// TwinCAT 3 PLC project tmo_spectrometer_motion
// ProgramVersion: 3.1.4022.7
// libraries:
//   lcls-twincat-motion, * (SLAC)
//   Tc2_MC2, * (Beckhoff Automation GmbH)
//   Tc2_Standard, * (Beckhoff Automation GmbH)
//   Tc2_System, * (Beckhoff Automation GmbH)
//   Tc2_Utilities, * (Beckhoff Automation GmbH)
//   Tc3_Module, * (Beckhoff Automation GmbH)
// project tree:
//   GVLs/ IO.TcGVL
//   / PlcTask.TcTTO
//   POUs/ Main.TcPOU
// real-time tasks:
//   TASK PlcTask: cycle T#10ms, priority 20, ADS port 350
// motion (NC):
//   TASK NC-Task 1 SAF: cycle T#2ms, priority 4, ADS port 501
//   TASK NC-Task 1 SVB: cycle T#10ms, priority 8, ADS port 511
//   AXIS LensX (id 1)
//     Dynamic: Acceleration=2, Deceleration=2
//     Velo: SlowManual=0.1, FastManual=1, Maximum=1
//     OtherSettings: AllowMotionCmdToSlave=true, PulseDistancePos=0.5, PulseDistanceNeg=0.5
//     encoder EncType=4
//       EncPara: ScaleFactorNumerator=3.90625e-05, MaxCount=#x0000ffff
//         Inc: RefSoftSyncMask=#x0000ffff
//     drive DrvType=24
//       Analog: VeloReferenz=4.5, ScaleFactorActTorque=0.1
//       TimeComp: TaskDelayCycles=1
//     controller CtrType=2
//       CtrPara: PriorControlFactor=1
//         PosDiffControl: Range=1
//         Observer: BandWidth=20
//   AXIS FoilX (id 2)
//     Dynamic: Acceleration=2, Deceleration=2
//     Velo: SlowManual=0.1, FastManual=1, Maximum=1
//     OtherSettings: AllowMotionCmdToSlave=true, PulseDistancePos=0.5, PulseDistanceNeg=0.5
//     encoder EncType=4
//       EncPara: ScaleFactorNumerator=0.000244140625, MaxCount=#x0000ffff
//         SoftEndMaxControl: Enable=true, Range=-1
//         Inc: RefSoftSyncMask=#x0000ffff
//     drive DrvType=24
//       Analog: VeloReferenz=31.25, ScaleFactorActTorque=0.1
//       TimeComp: TaskDelayCycles=1
//     controller CtrType=2
//       CtrPara: PriorControlFactor=1
//         PosDiffControl: Range=1
//         Observer: BandWidth=20
//   AXIS ZonePlateX (id 3)
//     Dynamic: Acceleration=2, Deceleration=2
//     Velo: SlowManual=0.1, FastManual=1, Maximum=1
//     OtherSettings: AllowMotionCmdToSlave=true, PulseDistancePos=0.5, PulseDistanceNeg=0.5
//     encoder EncType=4
//       EncPara: ScaleFactorNumerator=0.000103125, Inverse=true, MaxCount=#x0000ffff
//         Inc: RefSoftSyncMask=#x0000ffff
//     drive DrvType=24
//       DrvPara: Inverse=true
//         Analog: VeloReferenz=13.2, ScaleFactorActTorque=0.1
//         TimeComp: TaskDelayCycles=1
//     controller CtrType=2
//       CtrPara: PriorControlFactor=1
//         PosDiffControl: Range=1
//         Observer: BandWidth=20
//   AXIS ZonePlateY (id 4)
//     Dynamic: Acceleration=2, Deceleration=2
//     Velo: SlowManual=0.1, FastManual=1, Maximum=1
//     OtherSettings: AllowMotionCmdToSlave=true, PulseDistancePos=0.5, PulseDistanceNeg=0.5
//     encoder EncType=4
//       EncPara: ScaleFactorNumerator=4.6875e-05, MaxCount=#x0000ffff
//         Inc: RefSoftSyncMask=#x0000ffff
//     drive DrvType=24
//       Analog: VeloReferenz=6, ScaleFactorActTorque=0.1
//       TimeComp: TaskDelayCycles=1
//     controller CtrType=2
//       CtrPara: PriorControlFactor=1
//         PosDiffControl: Range=1
//         Observer: BandWidth=20
//   AXIS ZonePlateZ (id 5)
//     Dynamic: Acceleration=2, Deceleration=2
//     Velo: SlowManual=0.1, FastManual=1, Maximum=1
//     OtherSettings: AllowMotionCmdToSlave=true, PulseDistancePos=0.5, PulseDistanceNeg=0.5
//     encoder EncType=4
//       EncPara: ScaleFactorNumerator=7.8125e-05, ScaleFactorDenominator=1.6, MaxCount=#x0000ffff
//         Inc: RefSoftSyncMask=#x0000ffff
//     drive DrvType=24
//       Analog: VeloReferenz=6.25, ScaleFactorActTorque=0.1
//       TimeComp: TaskDelayCycles=1
//     controller CtrType=2
//       CtrPara: PriorControlFactor=1
//         PosDiffControl: Range=1
//         Observer: BandWidth=20
//   AXIS YagX (id 6)
//     Dynamic: Acceleration=2, Deceleration=2
//     Velo: SlowManual=0.1, FastManual=1, Maximum=1
//     OtherSettings: AllowMotionCmdToSlave=true, PulseDistancePos=0.5, PulseDistanceNeg=0.5
//     encoder EncType=4
//       EncPara: ScaleFactorNumerator=7.8125e-05, Inverse=true, MaxCount=#x0000ffff
//         Inc: RefSoftSyncMask=#x0000ffff
//     drive DrvType=24
//       DrvPara: Inverse=true
//         Analog: VeloReferenz=10, ScaleFactorActTorque=0.1
//         TimeComp: TaskDelayCycles=1
//     controller CtrType=2
//       CtrPara: PriorControlFactor=1
//         PosDiffControl: Range=1
//         Observer: BandWidth=20
//   AXIS YagY (id 7)
//     Dynamic: Acceleration=2, Deceleration=2
//     Velo: SlowManual=0.1, FastManual=1, Maximum=1
//     OtherSettings: AllowMotionCmdToSlave=true, PulseDistancePos=0.5, PulseDistanceNeg=0.5
//     encoder EncType=4
//       EncPara: ScaleFactorNumerator=7.8125e-05, MaxCount=#x0000ffff
//         Inc: RefSoftSyncMask=#x0000ffff
//     drive DrvType=24
//       Analog: VeloReferenz=10, ScaleFactorActTorque=0.1
//       TimeComp: TaskDelayCycles=1
//     controller CtrType=2
//       CtrPara: PriorControlFactor=1
//         PosDiffControl: Range=1
//         Observer: BandWidth=20
//   AXIS YagZ (id 8)
//     Dynamic: Acceleration=2, Deceleration=2
//     Velo: SlowManual=0.1, FastManual=1, Maximum=1
//     OtherSettings: AllowMotionCmdToSlave=true, PulseDistancePos=0.5, PulseDistanceNeg=0.5
//     encoder EncType=4
//       EncPara: ScaleFactorNumerator=9.6875e-05, Inverse=true, MaxCount=#x0000ffff
//         Inc: RefSoftSyncMask=#x0000ffff
//     drive DrvType=24
//       DrvPara: Inverse=true
//         Analog: VeloReferenz=12.7, ScaleFactorActTorque=0.1
//         TimeComp: TaskDelayCycles=1
//     controller CtrType=2
//       CtrPara: PriorControlFactor=1
//         PosDiffControl: Range=1
//         Observer: BandWidth=20
//   AXIS YagTheta (id 9)
//     Dynamic: Acceleration=2, Deceleration=2
//     Velo: SlowManual=0.1, FastManual=1, Maximum=1
//     OtherSettings: AllowMotionCmdToSlave=true, PulseDistancePos=0.5, PulseDistanceNeg=0.5
//     encoder EncType=4
//       EncPara: ScaleFactorNumerator=1.171875e-05, ScaleFactorDenominator=0.036667, MaxCount=#x0000ffff
//         Inc: RefSoftSyncMask=#x0000ffff
//     drive DrvType=24
//       Analog: VeloReferenz=409.0905372, ScaleFactorActTorque=0.1
//       TimeComp: TaskDelayCycles=1
//     controller CtrType=2
//       CtrPara: PriorControlFactor=1
//         PosDiffControl: Range=1
//         Observer: BandWidth=20
// I/O:
//   DEVICE Device 1 (EtherCAT), AmsNetId 172.21.132.142.2.1
//     Term 19 (EK1200) [EK1200-5000 EtherCAT Power supply (2A E-Bus)]
//       Term 20 (EL2202) [EL2202 2Ch. Dig. Output 24V, 0.5A]
//       Term 21 (EL6070) [EL6070 1Ch. Licensing-Terminal]
//       Term 22 (EL6695) [EL6695 EtherCAT Bridge terminal (Primary)]
//       Term 23 (EK1122) [EK1122 2 port EtherCAT junction]
//         Term 24 (EK1100) [EK1100 EtherCAT Coupler (2A E-Bus)]
//           EL7031-LensX [EL7031 1Ch. Stepper motor output stage (24V, 1.5A)]
//           LensX_EL1004
//           FoilX-EL7041 [EL7041 1Ch. Stepper motor output stage (50V, 5A)]
//           ZonePlateX-EL7041 [EL7041 1Ch. Stepper motor output stage (50V, 5A)]
//           ZonePlateY-EL7041 [EL7041 1Ch. Stepper motor output stage (50V, 5A)]
//           ZonePlateZ-EL7041 [EL7041 1Ch. Stepper motor output stage (50V, 5A)]
//           YagX-EL7041 [EL7041 1Ch. Stepper motor output stage (50V, 5A)]
//           YagY-EL7041 [EL7041 1Ch. Stepper motor output stage (50V, 5A)]
//           YagZ-EL7041 [EL7041 1Ch. Stepper motor output stage (50V, 5A)]
//           YagTheta-EL7041 [EL7041 1Ch. Stepper motor output stage (50V, 5A)]
//           Term 35 (EL9011) [EL9011 End Terminal]
// variable links:
//   (this object) <-> Device 1 (EtherCAT)/Term 19 (EK1200)/Term 23 (EK1122)/Term 24 (EK1100)/EL7031-LensX
//     Drive/Inputs/In/nState1 @bit 3 <-> STM Status/Status/Error
//     Drive/Inputs/In/nState1 @bit 5 <-> STM Status/Status/Moving negative
//     Drive/Inputs/In/nState1 @bit 4 <-> STM Status/Status/Moving positive
//     Drive/Inputs/In/nState1 @bit 1 <-> STM Status/Status/Ready
//     Drive/Inputs/In/nState1 <-> STM Status/Status/Ready to enable
//     Drive/Inputs/In/nState1 @bit 6 <-> STM Status/Status/Torque reduced
//     Drive/Inputs/In/nState1 @bit 2 <-> STM Status/Status/Warning
//     Drive/Inputs/In/nState2 @bit 3 <-> STM Status/Status/Digital input 1
//     Drive/Inputs/In/nState2 @bit 4 <-> STM Status/Status/Digital input 2
//     Drive/Inputs/In/nState2 @bit 5 <-> STM Status/Status/Sync error
//     Drive/Inputs/In/nState2 @bit 7 <-> STM Status/Status/TxPDO Toggle
//     Drive/Inputs/In/nState4 @bit 1 <-> WcState/InputToggle
//     Drive/Inputs/In/nState4 <-> WcState/WcState
//     Drive/Outputs/Out/nCtrl1 <-> STM Control/Control/Enable
//     Drive/Outputs/Out/nCtrl1 @bit 2 <-> STM Control/Control/Reduce torque
//     Drive/Outputs/Out/nCtrl1 @bit 1 <-> STM Control/Control/Reset
//     Drive/Outputs/Out/nDataOut2[0] <-> STM Velocity/Velocity
//     Enc/Inputs/In/nDataIn1[0] <-> ENC Status compact/Counter value
//     Enc/Inputs/In/nDataIn2[0] <-> ENC Status compact/Latch value
//     Enc/Inputs/In/nState1 @bit 4 <-> ENC Status compact/Status/Counter overflow
//     Enc/Inputs/In/nState1 @bit 3 <-> ENC Status compact/Status/Counter underflow
//     Enc/Inputs/In/nState1 @bit 1 <-> ENC Status compact/Status/Latch extern valid
//     Enc/Inputs/In/nState1 @bit 2 <-> ENC Status compact/Status/Set counter done
//     Enc/Inputs/In/nState2 @bit 4 <-> ENC Status compact/Status/Status of extern latch
//     Enc/Inputs/In/nState2 @bit 5 <-> ENC Status compact/Status/Sync error
//     Enc/Inputs/In/nState2 @bit 7 <-> ENC Status compact/Status/TxPDO Toggle
//     Enc/Inputs/In/nState4 @bit 1 <-> WcState/InputToggle
//     Enc/Inputs/In/nState4 <-> WcState/WcState
//     Enc/Outputs/Out/nCtrl1 @bit 3 <-> ENC Control compact/Control/Enable latch extern on negative edge
//     Enc/Outputs/Out/nCtrl1 @bit 1 <-> ENC Control compact/Control/Enable latch extern on positive edge
//     Enc/Outputs/Out/nCtrl1 @bit 2 <-> ENC Control compact/Control/Set counter
//     Enc/Outputs/Out/nDataOut1[0] <-> ENC Control compact/Set counter value
//   (this object) <-> Device 1 (EtherCAT)/Term 19 (EK1200)/Term 23 (EK1122)/Term 24 (EK1100)/FoilX-EL7041
//     Drive/Inputs/In/nState1 @bit 3 <-> STM Status/Status/Error
//     Drive/Inputs/In/nState1 @bit 5 <-> STM Status/Status/Moving negative
//     Drive/Inputs/In/nState1 @bit 4 <-> STM Status/Status/Moving positive
//     Drive/Inputs/In/nState1 @bit 1 <-> STM Status/Status/Ready
//     Drive/Inputs/In/nState1 <-> STM Status/Status/Ready to enable
//     Drive/Inputs/In/nState1 @bit 6 <-> STM Status/Status/Torque reduced
//     Drive/Inputs/In/nState1 @bit 2 <-> STM Status/Status/Warning
//     Drive/Inputs/In/nState2 @bit 3 <-> STM Status/Status/Digital input 1
//     Drive/Inputs/In/nState2 @bit 4 <-> STM Status/Status/Digital input 2
//     Drive/Inputs/In/nState2 @bit 5 <-> STM Status/Status/Sync error
//     Drive/Inputs/In/nState2 @bit 7 <-> STM Status/Status/TxPDO Toggle
//     Drive/Inputs/In/nState4 @bit 1 <-> WcState/InputToggle
//     Drive/Inputs/In/nState4 <-> WcState/WcState
//     Drive/Outputs/Out/nCtrl1 <-> STM Control/Control/Enable
//     Drive/Outputs/Out/nCtrl1 @bit 2 <-> STM Control/Control/Reduce torque
//     Drive/Outputs/Out/nCtrl1 @bit 1 <-> STM Control/Control/Reset
//     Drive/Outputs/Out/nDataOut2[0] <-> STM Velocity/Velocity
//     Enc/Inputs/In/nDataIn1[0] <-> ENC Status compact/Counter value
//     Enc/Inputs/In/nDataIn2[0] <-> ENC Status compact/Latch value
//     Enc/Inputs/In/nState1 @bit 4 <-> ENC Status compact/Status/Counter overflow
//     Enc/Inputs/In/nState1 @bit 3 <-> ENC Status compact/Status/Counter underflow
//     Enc/Inputs/In/nState1 @bit 7 <-> ENC Status compact/Status/Extrapolation stall
//     Enc/Inputs/In/nState1 <-> ENC Status compact/Status/Latch C valid
//     Enc/Inputs/In/nState1 @bit 1 <-> ENC Status compact/Status/Latch extern valid
//     Enc/Inputs/In/nState1 @bit 2 <-> ENC Status compact/Status/Set counter done
//     Enc/Inputs/In/nState2 @bit 4 <-> ENC Status compact/Status/Status of extern latch
//     Enc/Inputs/In/nState2 <-> ENC Status compact/Status/Status of input A
//     Enc/Inputs/In/nState2 @bit 1 <-> ENC Status compact/Status/Status of input B
//     Enc/Inputs/In/nState2 @bit 2 <-> ENC Status compact/Status/Status of input C
//     Enc/Inputs/In/nState2 @bit 5 <-> ENC Status compact/Status/Sync error
//     Enc/Inputs/In/nState2 @bit 7 <-> ENC Status compact/Status/TxPDO Toggle
//     Enc/Inputs/In/nState4 @bit 1 <-> WcState/InputToggle
//     Enc/Inputs/In/nState4 <-> WcState/WcState
//     Enc/Outputs/Out/nCtrl1 <-> ENC Control compact/Control/Enable latch C
//     Enc/Outputs/Out/nCtrl1 @bit 3 <-> ENC Control compact/Control/Enable latch extern on negative edge
//     Enc/Outputs/Out/nCtrl1 @bit 1 <-> ENC Control compact/Control/Enable latch extern on positive edge
//     Enc/Outputs/Out/nCtrl1 @bit 2 <-> ENC Control compact/Control/Set counter
//     Enc/Outputs/Out/nDataOut1[0] <-> ENC Control compact/Set counter value
//   (this object) <-> Device 1 (EtherCAT)/Term 19 (EK1200)/Term 23 (EK1122)/Term 24 (EK1100)/ZonePlateX-EL7041
//     Drive/Inputs/In/nState1 @bit 3 <-> STM Status/Status/Error
//     Drive/Inputs/In/nState1 @bit 5 <-> STM Status/Status/Moving negative
//     Drive/Inputs/In/nState1 @bit 4 <-> STM Status/Status/Moving positive
//     Drive/Inputs/In/nState1 @bit 1 <-> STM Status/Status/Ready
//     Drive/Inputs/In/nState1 <-> STM Status/Status/Ready to enable
//     Drive/Inputs/In/nState1 @bit 6 <-> STM Status/Status/Torque reduced
//     Drive/Inputs/In/nState1 @bit 2 <-> STM Status/Status/Warning
//     Drive/Inputs/In/nState2 @bit 3 <-> STM Status/Status/Digital input 1
//     Drive/Inputs/In/nState2 @bit 4 <-> STM Status/Status/Digital input 2
//     Drive/Inputs/In/nState2 @bit 5 <-> STM Status/Status/Sync error
//     Drive/Inputs/In/nState2 @bit 7 <-> STM Status/Status/TxPDO Toggle
//     Drive/Inputs/In/nState4 @bit 1 <-> WcState/InputToggle
//     Drive/Inputs/In/nState4 <-> WcState/WcState
//     Drive/Outputs/Out/nCtrl1 <-> STM Control/Control/Enable
//     Drive/Outputs/Out/nCtrl1 @bit 2 <-> STM Control/Control/Reduce torque
//     Drive/Outputs/Out/nCtrl1 @bit 1 <-> STM Control/Control/Reset
//     Drive/Outputs/Out/nDataOut2[0] <-> STM Velocity/Velocity
//     Enc/Inputs/In/nDataIn1[0] <-> ENC Status compact/Counter value
//     Enc/Inputs/In/nDataIn2[0] <-> ENC Status compact/Latch value
//     Enc/Inputs/In/nState1 @bit 4 <-> ENC Status compact/Status/Counter overflow
//     Enc/Inputs/In/nState1 @bit 3 <-> ENC Status compact/Status/Counter underflow
//     Enc/Inputs/In/nState1 @bit 7 <-> ENC Status compact/Status/Extrapolation stall
//     Enc/Inputs/In/nState1 <-> ENC Status compact/Status/Latch C valid
//     Enc/Inputs/In/nState1 @bit 1 <-> ENC Status compact/Status/Latch extern valid
//     Enc/Inputs/In/nState1 @bit 2 <-> ENC Status compact/Status/Set counter done
//     Enc/Inputs/In/nState2 @bit 4 <-> ENC Status compact/Status/Status of extern latch
//     Enc/Inputs/In/nState2 <-> ENC Status compact/Status/Status of input A
//     Enc/Inputs/In/nState2 @bit 1 <-> ENC Status compact/Status/Status of input B
//     Enc/Inputs/In/nState2 @bit 2 <-> ENC Status compact/Status/Status of input C
//     Enc/Inputs/In/nState2 @bit 5 <-> ENC Status compact/Status/Sync error
//     Enc/Inputs/In/nState2 @bit 7 <-> ENC Status compact/Status/TxPDO Toggle
//     Enc/Inputs/In/nState4 @bit 1 <-> WcState/InputToggle
//     Enc/Inputs/In/nState4 <-> WcState/WcState
//     Enc/Outputs/Out/nCtrl1 <-> ENC Control compact/Control/Enable latch C
//     Enc/Outputs/Out/nCtrl1 @bit 3 <-> ENC Control compact/Control/Enable latch extern on negative edge
//     Enc/Outputs/Out/nCtrl1 @bit 1 <-> ENC Control compact/Control/Enable latch extern on positive edge
//     Enc/Outputs/Out/nCtrl1 @bit 2 <-> ENC Control compact/Control/Set counter
//     Enc/Outputs/Out/nDataOut1[0] <-> ENC Control compact/Set counter value
//   (this object) <-> Device 1 (EtherCAT)/Term 19 (EK1200)/Term 23 (EK1122)/Term 24 (EK1100)/ZonePlateY-EL7041
//     Drive/Inputs/In/nState1 @bit 3 <-> STM Status/Status/Error
//     Drive/Inputs/In/nState1 @bit 5 <-> STM Status/Status/Moving negative
//     Drive/Inputs/In/nState1 @bit 4 <-> STM Status/Status/Moving positive
//     Drive/Inputs/In/nState1 @bit 1 <-> STM Status/Status/Ready
//     Drive/Inputs/In/nState1 <-> STM Status/Status/Ready to enable
//     Drive/Inputs/In/nState1 @bit 6 <-> STM Status/Status/Torque reduced
//     Drive/Inputs/In/nState1 @bit 2 <-> STM Status/Status/Warning
//     Drive/Inputs/In/nState2 @bit 3 <-> STM Status/Status/Digital input 1
//     Drive/Inputs/In/nState2 @bit 4 <-> STM Status/Status/Digital input 2
//     Drive/Inputs/In/nState2 @bit 5 <-> STM Status/Status/Sync error
//     Drive/Inputs/In/nState2 @bit 7 <-> STM Status/Status/TxPDO Toggle
//     Drive/Inputs/In/nState4 @bit 1 <-> WcState/InputToggle
//     Drive/Inputs/In/nState4 <-> WcState/WcState
//     Drive/Outputs/Out/nCtrl1 <-> STM Control/Control/Enable
//     Drive/Outputs/Out/nCtrl1 @bit 2 <-> STM Control/Control/Reduce torque
//     Drive/Outputs/Out/nCtrl1 @bit 1 <-> STM Control/Control/Reset
//     Drive/Outputs/Out/nDataOut2[0] <-> STM Velocity/Velocity
//     Enc/Inputs/In/nDataIn1[0] <-> ENC Status compact/Counter value
//     Enc/Inputs/In/nDataIn2[0] <-> ENC Status compact/Latch value
//     Enc/Inputs/In/nState1 @bit 4 <-> ENC Status compact/Status/Counter overflow
//     Enc/Inputs/In/nState1 @bit 3 <-> ENC Status compact/Status/Counter underflow
//     Enc/Inputs/In/nState1 @bit 7 <-> ENC Status compact/Status/Extrapolation stall
//     Enc/Inputs/In/nState1 <-> ENC Status compact/Status/Latch C valid
//     Enc/Inputs/In/nState1 @bit 1 <-> ENC Status compact/Status/Latch extern valid
//     Enc/Inputs/In/nState1 @bit 2 <-> ENC Status compact/Status/Set counter done
//     Enc/Inputs/In/nState2 @bit 4 <-> ENC Status compact/Status/Status of extern latch
//     Enc/Inputs/In/nState2 <-> ENC Status compact/Status/Status of input A
//     Enc/Inputs/In/nState2 @bit 1 <-> ENC Status compact/Status/Status of input B
//     Enc/Inputs/In/nState2 @bit 2 <-> ENC Status compact/Status/Status of input C
//     Enc/Inputs/In/nState2 @bit 5 <-> ENC Status compact/Status/Sync error
//     Enc/Inputs/In/nState2 @bit 7 <-> ENC Status compact/Status/TxPDO Toggle
//     Enc/Inputs/In/nState4 @bit 1 <-> WcState/InputToggle
//     Enc/Inputs/In/nState4 <-> WcState/WcState
//     Enc/Outputs/Out/nCtrl1 <-> ENC Control compact/Control/Enable latch C
//     Enc/Outputs/Out/nCtrl1 @bit 3 <-> ENC Control compact/Control/Enable latch extern on negative edge
//     Enc/Outputs/Out/nCtrl1 @bit 1 <-> ENC Control compact/Control/Enable latch extern on positive edge
//     Enc/Outputs/Out/nCtrl1 @bit 2 <-> ENC Control compact/Control/Set counter
//     Enc/Outputs/Out/nDataOut1[0] <-> ENC Control compact/Set counter value
//   (this object) <-> Device 1 (EtherCAT)/Term 19 (EK1200)/Term 23 (EK1122)/Term 24 (EK1100)/ZonePlateZ-EL7041
//     Drive/Inputs/In/nState1 @bit 3 <-> STM Status/Status/Error
//     Drive/Inputs/In/nState1 @bit 5 <-> STM Status/Status/Moving negative
//     Drive/Inputs/In/nState1 @bit 4 <-> STM Status/Status/Moving positive
//     Drive/Inputs/In/nState1 @bit 1 <-> STM Status/Status/Ready
//     Drive/Inputs/In/nState1 <-> STM Status/Status/Ready to enable
//     Drive/Inputs/In/nState1 @bit 6 <-> STM Status/Status/Torque reduced
//     Drive/Inputs/In/nState1 @bit 2 <-> STM Status/Status/Warning
//     Drive/Inputs/In/nState2 @bit 3 <-> STM Status/Status/Digital input 1
//     Drive/Inputs/In/nState2 @bit 4 <-> STM Status/Status/Digital input 2
//     Drive/Inputs/In/nState2 @bit 5 <-> STM Status/Status/Sync error
//     Drive/Inputs/In/nState2 @bit 7 <-> STM Status/Status/TxPDO Toggle
//     Drive/Inputs/In/nState4 @bit 1 <-> WcState/InputToggle
//     Drive/Inputs/In/nState4 <-> WcState/WcState
//     Drive/Outputs/Out/nCtrl1 <-> STM Control/Control/Enable
//     Drive/Outputs/Out/nCtrl1 @bit 2 <-> STM Control/Control/Reduce torque
//     Drive/Outputs/Out/nCtrl1 @bit 1 <-> STM Control/Control/Reset
//     Drive/Outputs/Out/nDataOut2[0] <-> STM Velocity/Velocity
//     Enc/Inputs/In/nDataIn1[0] <-> ENC Status compact/Counter value
//     Enc/Inputs/In/nDataIn2[0] <-> ENC Status compact/Latch value
//     Enc/Inputs/In/nState1 @bit 4 <-> ENC Status compact/Status/Counter overflow
//     Enc/Inputs/In/nState1 @bit 3 <-> ENC Status compact/Status/Counter underflow
//     Enc/Inputs/In/nState1 @bit 7 <-> ENC Status compact/Status/Extrapolation stall
//     Enc/Inputs/In/nState1 <-> ENC Status compact/Status/Latch C valid
//     Enc/Inputs/In/nState1 @bit 1 <-> ENC Status compact/Status/Latch extern valid
//     Enc/Inputs/In/nState1 @bit 2 <-> ENC Status compact/Status/Set counter done
//     Enc/Inputs/In/nState2 @bit 4 <-> ENC Status compact/Status/Status of extern latch
//     Enc/Inputs/In/nState2 <-> ENC Status compact/Status/Status of input A
//     Enc/Inputs/In/nState2 @bit 1 <-> ENC Status compact/Status/Status of input B
//     Enc/Inputs/In/nState2 @bit 2 <-> ENC Status compact/Status/Status of input C
//     Enc/Inputs/In/nState2 @bit 5 <-> ENC Status compact/Status/Sync error
//     Enc/Inputs/In/nState2 @bit 7 <-> ENC Status compact/Status/TxPDO Toggle
//     Enc/Inputs/In/nState4 @bit 1 <-> WcState/InputToggle
//     Enc/Inputs/In/nState4 <-> WcState/WcState
//     Enc/Outputs/Out/nCtrl1 <-> ENC Control compact/Control/Enable latch C
//     Enc/Outputs/Out/nCtrl1 @bit 3 <-> ENC Control compact/Control/Enable latch extern on negative edge
//     Enc/Outputs/Out/nCtrl1 @bit 1 <-> ENC Control compact/Control/Enable latch extern on positive edge
//     Enc/Outputs/Out/nCtrl1 @bit 2 <-> ENC Control compact/Control/Set counter
//     Enc/Outputs/Out/nDataOut1[0] <-> ENC Control compact/Set counter value
//   (this object) <-> Device 1 (EtherCAT)/Term 19 (EK1200)/Term 23 (EK1122)/Term 24 (EK1100)/YagX-EL7041
//     Drive/Inputs/In/nState1 @bit 3 <-> STM Status/Status/Error
//     Drive/Inputs/In/nState1 @bit 5 <-> STM Status/Status/Moving negative
//     Drive/Inputs/In/nState1 @bit 4 <-> STM Status/Status/Moving positive
//     Drive/Inputs/In/nState1 @bit 1 <-> STM Status/Status/Ready
//     Drive/Inputs/In/nState1 <-> STM Status/Status/Ready to enable
//     Drive/Inputs/In/nState1 @bit 6 <-> STM Status/Status/Torque reduced
//     Drive/Inputs/In/nState1 @bit 2 <-> STM Status/Status/Warning
//     Drive/Inputs/In/nState2 @bit 3 <-> STM Status/Status/Digital input 1
//     Drive/Inputs/In/nState2 @bit 4 <-> STM Status/Status/Digital input 2
//     Drive/Inputs/In/nState2 @bit 5 <-> STM Status/Status/Sync error
//     Drive/Inputs/In/nState2 @bit 7 <-> STM Status/Status/TxPDO Toggle
//     Drive/Inputs/In/nState4 @bit 1 <-> WcState/InputToggle
//     Drive/Inputs/In/nState4 <-> WcState/WcState
//     Drive/Outputs/Out/nCtrl1 <-> STM Control/Control/Enable
//     Drive/Outputs/Out/nCtrl1 @bit 2 <-> STM Control/Control/Reduce torque
//     Drive/Outputs/Out/nCtrl1 @bit 1 <-> STM Control/Control/Reset
//     Drive/Outputs/Out/nDataOut2[0] <-> STM Velocity/Velocity
//     Enc/Inputs/In/nDataIn1[0] <-> ENC Status compact/Counter value
//     Enc/Inputs/In/nDataIn2[0] <-> ENC Status compact/Latch value
//     Enc/Inputs/In/nState1 @bit 4 <-> ENC Status compact/Status/Counter overflow
//     Enc/Inputs/In/nState1 @bit 3 <-> ENC Status compact/Status/Counter underflow
//     Enc/Inputs/In/nState1 @bit 7 <-> ENC Status compact/Status/Extrapolation stall
//     Enc/Inputs/In/nState1 <-> ENC Status compact/Status/Latch C valid
//     Enc/Inputs/In/nState1 @bit 1 <-> ENC Status compact/Status/Latch extern valid
//     Enc/Inputs/In/nState1 @bit 2 <-> ENC Status compact/Status/Set counter done
//     Enc/Inputs/In/nState2 @bit 4 <-> ENC Status compact/Status/Status of extern latch
//     Enc/Inputs/In/nState2 <-> ENC Status compact/Status/Status of input A
//     Enc/Inputs/In/nState2 @bit 1 <-> ENC Status compact/Status/Status of input B
//     Enc/Inputs/In/nState2 @bit 2 <-> ENC Status compact/Status/Status of input C
//     Enc/Inputs/In/nState2 @bit 5 <-> ENC Status compact/Status/Sync error
//     Enc/Inputs/In/nState2 @bit 7 <-> ENC Status compact/Status/TxPDO Toggle
//     Enc/Inputs/In/nState4 @bit 1 <-> WcState/InputToggle
//     Enc/Inputs/In/nState4 <-> WcState/WcState
//     Enc/Outputs/Out/nCtrl1 <-> ENC Control compact/Control/Enable latch C
//     Enc/Outputs/Out/nCtrl1 @bit 3 <-> ENC Control compact/Control/Enable latch extern on negative edge
//     Enc/Outputs/Out/nCtrl1 @bit 1 <-> ENC Control compact/Control/Enable latch extern on positive edge
//     Enc/Outputs/Out/nCtrl1 @bit 2 <-> ENC Control compact/Control/Set counter
//     Enc/Outputs/Out/nDataOut1[0] <-> ENC Control compact/Set counter value
//   (this object) <-> Device 1 (EtherCAT)/Term 19 (EK1200)/Term 23 (EK1122)/Term 24 (EK1100)/YagY-EL7041
//     Drive/Inputs/In/nState1 @bit 3 <-> STM Status/Status/Error
//     Drive/Inputs/In/nState1 @bit 5 <-> STM Status/Status/Moving negative
//     Drive/Inputs/In/nState1 @bit 4 <-> STM Status/Status/Moving positive
//     Drive/Inputs/In/nState1 @bit 1 <-> STM Status/Status/Ready
//     Drive/Inputs/In/nState1 <-> STM Status/Status/Ready to enable
//     Drive/Inputs/In/nState1 @bit 6 <-> STM Status/Status/Torque reduced
//     Drive/Inputs/In/nState1 @bit 2 <-> STM Status/Status/Warning
//     Drive/Inputs/In/nState2 @bit 3 <-> STM Status/Status/Digital input 1
//     Drive/Inputs/In/nState2 @bit 4 <-> STM Status/Status/Digital input 2
//     Drive/Inputs/In/nState2 @bit 5 <-> STM Status/Status/Sync error
//     Drive/Inputs/In/nState2 @bit 7 <-> STM Status/Status/TxPDO Toggle
//     Drive/Inputs/In/nState4 @bit 1 <-> WcState/InputToggle
//     Drive/Inputs/In/nState4 <-> WcState/WcState
//     Drive/Outputs/Out/nCtrl1 <-> STM Control/Control/Enable
//     Drive/Outputs/Out/nCtrl1 @bit 2 <-> STM Control/Control/Reduce torque
//     Drive/Outputs/Out/nCtrl1 @bit 1 <-> STM Control/Control/Reset
//     Drive/Outputs/Out/nDataOut2[0] <-> STM Velocity/Velocity
//     Enc/Inputs/In/nDataIn1[0] <-> ENC Status compact/Counter value
//     Enc/Inputs/In/nDataIn2[0] <-> ENC Status compact/Latch value
//     Enc/Inputs/In/nState1 @bit 4 <-> ENC Status compact/Status/Counter overflow
//     Enc/Inputs/In/nState1 @bit 3 <-> ENC Status compact/Status/Counter underflow
//     Enc/Inputs/In/nState1 @bit 7 <-> ENC Status compact/Status/Extrapolation stall
//     Enc/Inputs/In/nState1 <-> ENC Status compact/Status/Latch C valid
//     Enc/Inputs/In/nState1 @bit 1 <-> ENC Status compact/Status/Latch extern valid
//     Enc/Inputs/In/nState1 @bit 2 <-> ENC Status compact/Status/Set counter done
//     Enc/Inputs/In/nState2 @bit 4 <-> ENC Status compact/Status/Status of extern latch
//     Enc/Inputs/In/nState2 <-> ENC Status compact/Status/Status of input A
//     Enc/Inputs/In/nState2 @bit 1 <-> ENC Status compact/Status/Status of input B
//     Enc/Inputs/In/nState2 @bit 2 <-> ENC Status compact/Status/Status of input C
//     Enc/Inputs/In/nState2 @bit 5 <-> ENC Status compact/Status/Sync error
//     Enc/Inputs/In/nState2 @bit 7 <-> ENC Status compact/Status/TxPDO Toggle
//     Enc/Inputs/In/nState4 @bit 1 <-> WcState/InputToggle
//     Enc/Inputs/In/nState4 <-> WcState/WcState
//     Enc/Outputs/Out/nCtrl1 <-> ENC Control compact/Control/Enable latch C
//     Enc/Outputs/Out/nCtrl1 @bit 3 <-> ENC Control compact/Control/Enable latch extern on negative edge
//     Enc/Outputs/Out/nCtrl1 @bit 1 <-> ENC Control compact/Control/Enable latch extern on positive edge
//     Enc/Outputs/Out/nCtrl1 @bit 2 <-> ENC Control compact/Control/Set counter
//     Enc/Outputs/Out/nDataOut1[0] <-> ENC Control compact/Set counter value
//   (this object) <-> Device 1 (EtherCAT)/Term 19 (EK1200)/Term 23 (EK1122)/Term 24 (EK1100)/YagZ-EL7041
//     Drive/Inputs/In/nState1 @bit 3 <-> STM Status/Status/Error
//     Drive/Inputs/In/nState1 @bit 5 <-> STM Status/Status/Moving negative
//     Drive/Inputs/In/nState1 @bit 4 <-> STM Status/Status/Moving positive
//     Drive/Inputs/In/nState1 @bit 1 <-> STM Status/Status/Ready
//     Drive/Inputs/In/nState1 <-> STM Status/Status/Ready to enable
//     Drive/Inputs/In/nState1 @bit 6 <-> STM Status/Status/Torque reduced
//     Drive/Inputs/In/nState1 @bit 2 <-> STM Status/Status/Warning
//     Drive/Inputs/In/nState2 @bit 3 <-> STM Status/Status/Digital input 1
//     Drive/Inputs/In/nState2 @bit 4 <-> STM Status/Status/Digital input 2
//     Drive/Inputs/In/nState2 @bit 5 <-> STM Status/Status/Sync error
//     Drive/Inputs/In/nState2 @bit 7 <-> STM Status/Status/TxPDO Toggle
//     Drive/Inputs/In/nState4 @bit 1 <-> WcState/InputToggle
//     Drive/Inputs/In/nState4 <-> WcState/WcState
//     Drive/Outputs/Out/nCtrl1 <-> STM Control/Control/Enable
//     Drive/Outputs/Out/nCtrl1 @bit 2 <-> STM Control/Control/Reduce torque
//     Drive/Outputs/Out/nCtrl1 @bit 1 <-> STM Control/Control/Reset
//     Drive/Outputs/Out/nDataOut2[0] <-> STM Velocity/Velocity
//     Enc/Inputs/In/nDataIn1[0] <-> ENC Status compact/Counter value
//     Enc/Inputs/In/nDataIn2[0] <-> ENC Status compact/Latch value
//     Enc/Inputs/In/nState1 @bit 4 <-> ENC Status compact/Status/Counter overflow
//     Enc/Inputs/In/nState1 @bit 3 <-> ENC Status compact/Status/Counter underflow
//     Enc/Inputs/In/nState1 @bit 7 <-> ENC Status compact/Status/Extrapolation stall
//     Enc/Inputs/In/nState1 <-> ENC Status compact/Status/Latch C valid
//     Enc/Inputs/In/nState1 @bit 1 <-> ENC Status compact/Status/Latch extern valid
//     Enc/Inputs/In/nState1 @bit 2 <-> ENC Status compact/Status/Set counter done
//     Enc/Inputs/In/nState2 @bit 4 <-> ENC Status compact/Status/Status of extern latch
//     Enc/Inputs/In/nState2 <-> ENC Status compact/Status/Status of input A
//     Enc/Inputs/In/nState2 @bit 1 <-> ENC Status compact/Status/Status of input B
//     Enc/Inputs/In/nState2 @bit 2 <-> ENC Status compact/Status/Status of input C
//     Enc/Inputs/In/nState2 @bit 5 <-> ENC Status compact/Status/Sync error
//     Enc/Inputs/In/nState2 @bit 7 <-> ENC Status compact/Status/TxPDO Toggle
//     Enc/Inputs/In/nState4 @bit 1 <-> WcState/InputToggle
//     Enc/Inputs/In/nState4 <-> WcState/WcState
//     Enc/Outputs/Out/nCtrl1 <-> ENC Control compact/Control/Enable latch C
//     Enc/Outputs/Out/nCtrl1 @bit 3 <-> ENC Control compact/Control/Enable latch extern on negative edge
//     Enc/Outputs/Out/nCtrl1 @bit 1 <-> ENC Control compact/Control/Enable latch extern on positive edge
//     Enc/Outputs/Out/nCtrl1 @bit 2 <-> ENC Control compact/Control/Set counter
//     Enc/Outputs/Out/nDataOut1[0] <-> ENC Control compact/Set counter value
//   (this object) <-> Device 1 (EtherCAT)/Term 19 (EK1200)/Term 23 (EK1122)/Term 24 (EK1100)/YagTheta-EL7041
//     Drive/Inputs/In/nState1 @bit 3 <-> STM Status/Status/Error
//     Drive/Inputs/In/nState1 @bit 5 <-> STM Status/Status/Moving negative
//     Drive/Inputs/In/nState1 @bit 4 <-> STM Status/Status/Moving positive
//     Drive/Inputs/In/nState1 @bit 1 <-> STM Status/Status/Ready
//     Drive/Inputs/In/nState1 <-> STM Status/Status/Ready to enable
//     Drive/Inputs/In/nState1 @bit 6 <-> STM Status/Status/Torque reduced
//     Drive/Inputs/In/nState1 @bit 2 <-> STM Status/Status/Warning
//     Drive/Inputs/In/nState2 @bit 3 <-> STM Status/Status/Digital input 1
//     Drive/Inputs/In/nState2 @bit 4 <-> STM Status/Status/Digital input 2
//     Drive/Inputs/In/nState2 @bit 5 <-> STM Status/Status/Sync error
//     Drive/Inputs/In/nState2 @bit 7 <-> STM Status/Status/TxPDO Toggle
//     Drive/Inputs/In/nState4 @bit 1 <-> WcState/InputToggle
//     Drive/Inputs/In/nState4 <-> WcState/WcState
//     Drive/Outputs/Out/nCtrl1 <-> STM Control/Control/Enable
//     Drive/Outputs/Out/nCtrl1 @bit 2 <-> STM Control/Control/Reduce torque
//     Drive/Outputs/Out/nCtrl1 @bit 1 <-> STM Control/Control/Reset
//     Drive/Outputs/Out/nDataOut2[0] <-> STM Velocity/Velocity
//     Enc/Inputs/In/nDataIn1[0] <-> ENC Status compact/Counter value
//     Enc/Inputs/In/nDataIn2[0] <-> ENC Status compact/Latch value
//     Enc/Inputs/In/nState1 @bit 4 <-> ENC Status compact/Status/Counter overflow
//     Enc/Inputs/In/nState1 @bit 3 <-> ENC Status compact/Status/Counter underflow
//     Enc/Inputs/In/nState1 @bit 7 <-> ENC Status compact/Status/Extrapolation stall
//     Enc/Inputs/In/nState1 <-> ENC Status compact/Status/Latch C valid
//     Enc/Inputs/In/nState1 @bit 1 <-> ENC Status compact/Status/Latch extern valid
//     Enc/Inputs/In/nState1 @bit 2 <-> ENC Status compact/Status/Set counter done
//     Enc/Inputs/In/nState2 @bit 4 <-> ENC Status compact/Status/Status of extern latch
//     Enc/Inputs/In/nState2 <-> ENC Status compact/Status/Status of input A
//     Enc/Inputs/In/nState2 @bit 1 <-> ENC Status compact/Status/Status of input B
//     Enc/Inputs/In/nState2 @bit 2 <-> ENC Status compact/Status/Status of input C
//     Enc/Inputs/In/nState2 @bit 5 <-> ENC Status compact/Status/Sync error
//     Enc/Inputs/In/nState2 @bit 7 <-> ENC Status compact/Status/TxPDO Toggle
//     Enc/Inputs/In/nState4 @bit 1 <-> WcState/InputToggle
//     Enc/Inputs/In/nState4 <-> WcState/WcState
//     Enc/Outputs/Out/nCtrl1 <-> ENC Control compact/Control/Enable latch C
//     Enc/Outputs/Out/nCtrl1 @bit 3 <-> ENC Control compact/Control/Enable latch extern on negative edge
//     Enc/Outputs/Out/nCtrl1 @bit 1 <-> ENC Control compact/Control/Enable latch extern on positive edge
//     Enc/Outputs/Out/nCtrl1 @bit 2 <-> ENC Control compact/Control/Set counter
//     Enc/Outputs/Out/nDataOut1[0] <-> ENC Control compact/Set counter value
//   tmo_spectrometer_motion Instance <-> Device 1 (EtherCAT)/Term 19 (EK1200)/Term 23 (EK1122)/Term 24 (EK1100)/FoilX-EL7041
//     PlcTask Inputs/Main.M2.bLimitBackwardEnable <-> STM Status/Status/Digital input 2
//     PlcTask Inputs/Main.M2.bLimitForwardEnable <-> STM Status/Status/Digital input 1
//   tmo_spectrometer_motion Instance <-> Device 1 (EtherCAT)/Term 19 (EK1200)/Term 23 (EK1122)/Term 24 (EK1100)/LensX_EL1004
//     PlcTask Inputs/IO.bMyInput1 <-> Channel 1/Input
//     PlcTask Inputs/IO.bMyInput2 <-> Channel 2/Input
//   tmo_spectrometer_motion Instance <-> Device 1 (EtherCAT)/Term 19 (EK1200)/Term 23 (EK1122)/Term 24 (EK1100)/YagTheta-EL7041
//     PlcTask Inputs/Main.M9.bLimitBackwardEnable <-> STM Status/Status/Digital input 2
//     PlcTask Inputs/Main.M9.bLimitForwardEnable <-> STM Status/Status/Digital input 1
//   tmo_spectrometer_motion Instance <-> Device 1 (EtherCAT)/Term 19 (EK1200)/Term 23 (EK1122)/Term 24 (EK1100)/YagX-EL7041
//     PlcTask Inputs/Main.M6.bLimitBackwardEnable <-> STM Status/Status/Digital input 1
//     PlcTask Inputs/Main.M6.bLimitForwardEnable <-> STM Status/Status/Digital input 2
//   tmo_spectrometer_motion Instance <-> Device 1 (EtherCAT)/Term 19 (EK1200)/Term 23 (EK1122)/Term 24 (EK1100)/YagY-EL7041
//     PlcTask Inputs/Main.M7.bLimitBackwardEnable <-> STM Status/Status/Digital input 2
//     PlcTask Inputs/Main.M7.bLimitForwardEnable <-> STM Status/Status/Digital input 1
//   tmo_spectrometer_motion Instance <-> Device 1 (EtherCAT)/Term 19 (EK1200)/Term 23 (EK1122)/Term 24 (EK1100)/YagZ-EL7041
//     PlcTask Inputs/Main.M8.bLimitBackwardEnable <-> STM Status/Status/Digital input 1
//     PlcTask Inputs/Main.M8.bLimitForwardEnable <-> STM Status/Status/Digital input 2
//   tmo_spectrometer_motion Instance <-> Device 1 (EtherCAT)/Term 19 (EK1200)/Term 23 (EK1122)/Term 24 (EK1100)/ZonePlateX-EL7041
//     PlcTask Inputs/Main.M3.bLimitBackwardEnable <-> STM Status/Status/Digital input 1
//     PlcTask Inputs/Main.M3.bLimitForwardEnable <-> STM Status/Status/Digital input 2
//   tmo_spectrometer_motion Instance <-> Device 1 (EtherCAT)/Term 19 (EK1200)/Term 23 (EK1122)/Term 24 (EK1100)/ZonePlateY-EL7041
//     PlcTask Inputs/Main.M4.bLimitBackwardEnable <-> STM Status/Status/Digital input 1
//     PlcTask Inputs/Main.M4.bLimitForwardEnable <-> STM Status/Status/Digital input 2
//   tmo_spectrometer_motion Instance <-> Device 1 (EtherCAT)/Term 19 (EK1200)/Term 23 (EK1122)/Term 24 (EK1100)/ZonePlateZ-EL7041
//     PlcTask Inputs/Main.M5.bLimitBackwardEnable <-> STM Status/Status/Digital input 2
//     PlcTask Inputs/Main.M5.bLimitForwardEnable <-> STM Status/Status/Digital input 1
//   tmo_spectrometer_motion Instance <-> NC-Task 1 SAF/Axes/FoilX
//     PlcTask Inputs/Main.M2.Axis.NcToPlc <-> Outputs/ToPlc
//     PlcTask Outputs/Main.M2.Axis.PlcToNc <-> Inputs/FromPlc
//   tmo_spectrometer_motion Instance <-> NC-Task 1 SAF/Axes/LensX
//     PlcTask Inputs/Main.M1.Axis.NcToPlc <-> Outputs/ToPlc
//     PlcTask Outputs/Main.M1.Axis.PlcToNc <-> Inputs/FromPlc
//   tmo_spectrometer_motion Instance <-> NC-Task 1 SAF/Axes/YagTheta
//     PlcTask Inputs/Main.M9.Axis.NcToPlc <-> Outputs/ToPlc
//     PlcTask Outputs/Main.M9.Axis.PlcToNc <-> Inputs/FromPlc
//   tmo_spectrometer_motion Instance <-> NC-Task 1 SAF/Axes/YagX
//     PlcTask Inputs/Main.M6.Axis.NcToPlc <-> Outputs/ToPlc
//     PlcTask Outputs/Main.M6.Axis.PlcToNc <-> Inputs/FromPlc
//   tmo_spectrometer_motion Instance <-> NC-Task 1 SAF/Axes/YagY
//     PlcTask Inputs/Main.M7.Axis.NcToPlc <-> Outputs/ToPlc
//     PlcTask Outputs/Main.M7.Axis.PlcToNc <-> Inputs/FromPlc
//   tmo_spectrometer_motion Instance <-> NC-Task 1 SAF/Axes/YagZ
//     PlcTask Inputs/Main.M8.Axis.NcToPlc <-> Outputs/ToPlc
//     PlcTask Outputs/Main.M8.Axis.PlcToNc <-> Inputs/FromPlc
//   tmo_spectrometer_motion Instance <-> NC-Task 1 SAF/Axes/ZonePlateX
//     PlcTask Inputs/Main.M3.Axis.NcToPlc <-> Outputs/ToPlc
//     PlcTask Outputs/Main.M3.Axis.PlcToNc <-> Inputs/FromPlc
//   tmo_spectrometer_motion Instance <-> NC-Task 1 SAF/Axes/ZonePlateY
//     PlcTask Inputs/Main.M4.Axis.NcToPlc <-> Outputs/ToPlc
//     PlcTask Outputs/Main.M4.Axis.PlcToNc <-> Inputs/FromPlc
//   tmo_spectrometer_motion Instance <-> NC-Task 1 SAF/Axes/ZonePlateZ
//     PlcTask Inputs/Main.M5.Axis.NcToPlc <-> Outputs/ToPlc
//     PlcTask Outputs/Main.M5.Axis.PlcToNc <-> Inputs/FromPlc

CONFIGURATION tmo_spectrometer_motion
    RESOURCE PLC ON TwinCAT3
        TASK PlcTask(INTERVAL := T#10ms, PRIORITY := 20);
        PROGRAM Main WITH PlcTask : Main;
    END_RESOURCE
END_CONFIGURATION

// ---- GVLs/IO.TcGVL
{attribute 'qualified_only'}
VAR_GLOBAL
	{attribute 'TcLinkTo' := 'TIID^Device 1 (EtherCAT)^Term 19 (EK1200)^Term 23 (EK1122)^Term 24 (EK1100)^LensX-EL1004^Channel 1^Input'}
	bMyInput1 AT %I* : BOOL;

	{attribute 'TcLinkTo' := 'TIID^Device 1 (EtherCAT)^Term 19 (EK1200)^Term 23 (EK1122)^Term 24 (EK1100)^LensX-EL1004^Channel 2^Input'}
	bMyInput2 AT %I* : BOOL;

END_VAR

// ---- POUs/Main.TcPOU
PROGRAM Main
VAR
    // Motors
    // Spectrometer Axes
//    {attribute 'TcLinkTo' := '.bMyInput1:=TIIB[LensX-EL1004]^Channel 1^Input;
//                             .bMyInput2:=TIIB[LensX-EL1004]^Channel 2^Input'}
    {attribute 'pytmc' := '
        pv: TMO:SPEC:MMS:01
    '}
	
    M1 : DUT_MotionStage := (bPowerSelf:=TRUE,
    nEnableMode:=ENUM_StageEnableMode.DURING_MOTION,
//    nEnableMode:=ENUM_StageEnableMode.ALWAYS,
    nHomingMode := ENUM_EpicsHomeCmd.ABSOLUTE_SET); // Lens X

    {attribute 'TcLinkTo' := '.bLimitForwardEnable:=TIIB[FoilX-EL7041]^STM Status^Status^Digital input 1;
                              .bLimitBackwardEnable:=TIIB[FoilX-EL7041]^STM Status^Status^Digital input 2'}
    {attribute 'pytmc' := '
        pv: TMO:SPEC:MMS:02
    '}
    M2 : DUT_MotionStage := (bPowerSelf:=TRUE,
	nEnableMode:=ENUM_StageEnableMode.DURING_MOTION,
//    nEnableMode:=ENUM_StageEnableMode.ALWAYS,
    nHomingMode := ENUM_EpicsHomeCmd.ABSOLUTE_SET); // AL Foil X

    {attribute 'TcLinkTo' := '.bLimitForwardEnable:=TIIB[ZonePlateX-EL7041]^STM Status^Status^Digital input 2;
                              .bLimitBackwardEnable:=TIIB[ZonePlateX-EL7041]^STM Status^Status^Digital input 1'}
    {attribute 'pytmc' := '
        pv: TMO:SPEC:MMS:03
    '}
    M3 : DUT_MotionStage := (bPowerSelf:=TRUE,
	nEnableMode:=ENUM_StageEnableMode.DURING_MOTION,
//    nEnableMode:=ENUM_StageEnableMode.ALWAYS,
    nHomingMode := ENUM_EpicsHomeCmd.ABSOLUTE_SET); // Zone Plate X

    {attribute 'TcLinkTo' := '.bLimitForwardEnable:=TIIB[ZonePlateY-EL7041]^STM Status^Status^Digital input 2;
                              .bLimitBackwardEnable:=TIIB[ZonePlateY-EL7041]^STM Status^Status^Digital input 1'}
    {attribute 'pytmc' := '
        pv: TMO:SPEC:MMS:04
    '}
    M4 : DUT_MotionStage := (bPowerSelf:=TRUE,
	nEnableMode:=ENUM_StageEnableMode.DURING_MOTION,
//    nEnableMode:=ENUM_StageEnableMode.ALWAYS,
    nHomingMode := ENUM_EpicsHomeCmd.ABSOLUTE_SET); // Zone Plate Y

    {attribute 'TcLinkTo' := '.bLimitForwardEnable:=TIIB[ZonePlateZ-EL7041]^STM Status^Status^Digital input 1;
                              .bLimitBackwardEnable:=TIIB[ZonePlateZ-EL7041]^STM Status^Status^Digital input 2'}
    {attribute 'pytmc' := '
        pv: TMO:SPEC:MMS:05
    '}
    M5 : DUT_MotionStage := (bPowerSelf:=TRUE,
	nEnableMode:=ENUM_StageEnableMode.DURING_MOTION,
//    nEnableMode:=ENUM_StageEnableMode.ALWAYS,
    nHomingMode := ENUM_EpicsHomeCmd.ABSOLUTE_SET); // Zone Plate Z

    {attribute 'TcLinkTo' := '.bLimitForwardEnable:=TIIB[YagX-EL7041]^STM Status^Status^Digital input 2;
                              .bLimitBackwardEnable:=TIIB[YagX-EL7041]^STM Status^Status^Digital input 1'}
    {attribute 'pytmc' := '
        pv: TMO:SPEC:MMS:06
    '}
    M6 : DUT_MotionStage := (bPowerSelf:=TRUE,
	nEnableMode:=ENUM_StageEnableMode.DURING_MOTION,
//    nEnableMode:=ENUM_StageEnableMode.ALWAYS,
    nHomingMode := ENUM_EpicsHomeCmd.ABSOLUTE_SET); // Yag X
	
    {attribute 'TcLinkTo' := '.bLimitForwardEnable:=TIIB[YagY-EL7041]^STM Status^Status^Digital input 1;
                              .bLimitBackwardEnable:=TIIB[YagY-EL7041]^STM Status^Status^Digital input 2'}
    {attribute 'pytmc' := '
        pv: TMO:SPEC:MMS:07
    '}
    M7 : DUT_MotionStage := (bPowerSelf:=TRUE,
	nEnableMode:=ENUM_StageEnableMode.DURING_MOTION,
//    nEnableMode:=ENUM_StageEnableMode.ALWAYS,
    nHomingMode := ENUM_EpicsHomeCmd.ABSOLUTE_SET); // Yag Y
	
	{attribute 'TcLinkTo' := '.bLimitForwardEnable:=TIIB[YagZ-EL7041]^STM Status^Status^Digital input 2;
                              .bLimitBackwardEnable:=TIIB[YagZ-EL7041]^STM Status^Status^Digital input 1'}
    {attribute 'pytmc' := '
        pv: TMO:SPEC:MMS:08
    '}
    M8 : DUT_MotionStage := (bPowerSelf:=TRUE,
	nEnableMode:=ENUM_StageEnableMode.DURING_MOTION,
//    nEnableMode:=ENUM_StageEnableMode.ALWAYS,
    nHomingMode := ENUM_EpicsHomeCmd.ABSOLUTE_SET); // Yag Z
	
	{attribute 'TcLinkTo' := '.bLimitForwardEnable:=TIIB[YagTheta-EL7041]^STM Status^Status^Digital input 1;
                              .bLimitBackwardEnable:=TIIB[YagTheta-EL7041]^STM Status^Status^Digital input 2'}
    {attribute 'pytmc' := '
        pv: TMO:SPEC:MMS:09
    '}
    M9 : DUT_MotionStage := (bPowerSelf:=TRUE,
	nEnableMode:=ENUM_StageEnableMode.DURING_MOTION,
//    nEnableMode:=ENUM_StageEnableMode.ALWAYS,
    nHomingMode := ENUM_EpicsHomeCmd.ABSOLUTE_SET); // Yag Theta
	
    // Spectrometer Axes
    fbMotionStageM1 : FB_MotionStage;
    fbMotionStageM2 : FB_MotionStage;
    fbMotionStageM3 : FB_MotionStage;
    fbMotionStageM4 : FB_MotionStage;
    fbMotionStageM5 : FB_MotionStage;
    fbMotionStageM6 : FB_MotionStage;
    fbMotionStageM7 : FB_MotionStage;               
    fbMotionStageM8 : FB_MotionStage;
    fbMotionStageM9 : FB_MotionStage;
	
//	motorlimit: BOOL;
//	bLimitForwardEnable: BOOL;
//	bMyInput: BOOL;
//	bMyInput2: BOOL;
//	bMyInput1: BOOL;
END_VAR
	(*
	// Persistent Memory
	fbWritePersistentData : WritePersistentData;
	bInit : BOOL := TRUE;
	fbWriteDelay : TON;
	mcSetPosition : ARRAY [1..6] of MC_SetPosition;

VAR PERSISTENT
	fLensXPos : LREAL;
	fFoilXPos : LREAL;
	fZonePlateXPos : LREAL;
	fZonePlateYPos : LREAL;
	fZonePlateZPos : LREAL;
	fYagXPos : LREAL;
END_VAR
*)

(*IF bInit THEN
	//Sets axes positions with persistent value
	// Gas Nozzle
	mcSetPosition[1](Axis:=M1.Axis, Position:=fLensXPos, Mode:=FALSE, Execute:=TRUE);
	mcSetPosition[2](Axis:=M2.Axis, Position:=fFoilXPos, Mode:=FALSE, Execute:=TRUE);
	mcSetPosition[3](Axis:=M3.Axis, Position:=fZonePlateXPos, Mode:=FALSE, Execute:=TRUE);
	// Sample Paddle
    mcSetPosition[4](Axis:=M4.Axis, Position:=fZonePlateYPos, Mode:=FALSE, Execute:=TRUE);
	mcSetPosition[5](Axis:=M5.Axis, Position:=fZonePlateZPos, Mode:=FALSE, Execute:=TRUE);
	mcSetPosition[6](Axis:=M6.Axis, Position:=fYagXPos, Mode:=FALSE, Execute:=TRUE);
    if(mcSetPosition[1].Done and NOT mcSetPosition[1].Error) AND 
      (mcSetPosition[2].Done and NOT mcSetPosition[2].Error) AND
	  (mcSetPosition[3].Done and NOT mcSetPosition[3].Error) AND
	  (mcSetPosition[4].Done and NOT mcSetPosition[4].Error) AND
	  (mcSetPosition[5].Done and NOT mcSetPosition[5].Error) AND
	  (mcSetPosition[6].Done and Not mcSetPosition[6].Error) THEN
	  bInit:=FALSE;
	  
	  mcSetPosition[1](Axis:=M1.Axis, Execute:=FALSE);
	  mcSetPosition[2](Axis:=M2.Axis, Execute:=FALSE);
	  mcSetPosition[3](Axis:=M3.Axis, Execute:=FALSE);
	  mcSetPosition[4](Axis:=M4.Axis, Execute:=FALSE);
	  mcSetPosition[5](Axis:=M5.Axis, Execute:=FALSE);
	  mcSetPosition[6](Axis:=M6.Axis, Execute:=FALSE);
	END_IF
ELSE
*)
// Hardware Enable and fbMotionStage
//Lens X
	M1.bHardwareEnable := TRUE;
	fbMotionStageM1(stMotionStage:=M1);
// AL Foil X
	M2.bHardwareEnable := TRUE;
	fbMotionStageM2(stMotionStage:=M2);
//Zone Plate
	M3.bHardwareEnable := TRUE;
	fbMotionStageM3(stMotionStage:=M3);
	
	M4.bHardwareEnable := TRUE;
	fbMotionStageM4(stMotionStage:=M4);

	M5.bHardwareEnable := TRUE;
	fbMotionStageM5(stMotionStage:=M5);
// YAG
	M6.bHardwareEnable := TRUE;
	fbMotionStageM6(stMotionStage:=M6);
	
	M7.bHardwareEnable := TRUE;
	fbMotionStageM7(stMotionStage:=M7);
	
	M8.bHardwareEnable := TRUE;
	fbMotionStageM8(stMotionStage:=M8);
	
	M9.bHardwareEnable := TRUE;
    fbMotionStageM9(stMotionStage:=M9);	
	
//    M1.bLimitForwardEnable:=not io.bMyInput;

    M1.bLimitForwardEnable:=not IO.bMyInput1;
	M1.bLimitBackwardEnable:=not IO.bMyInput2;
(*
// Keep track of position

	fLensXPos := M1.Axis.NcToPlc.ActPos;
	fFoilXPos := M2.Axis.NcToPlc.ActPos;
	fZonePlateXPos := M3.Axis.NcToPlc.ActPos;
	fZonePlateYPos := M4.Axis.NcToPlc.ActPos;
	fZonePlateZPos := M5.Axis.NcToPlc.ActPos;
	fYagXPos := M6.Axis.NcToPlc.ActPos;	

// Persistent Memory
	IF fbWriteDelay.Q THEN
		fbWritePersistentData(NETID:='', PORT:=851, START:=TRUE, TMOUT:=T#1S);
		fbWriteDelay(IN:=FALSE);
	ELSE
		fbWritePersistentData(START:=FALSE);
		fbWriteDelay(IN:=TRUE, PT:=T#0.5S);
	END_IF
END_IF;
*)

END_PROGRAM
